SUBAPPLICATION FillWindowFS_AR (* Färbt ein FillAttributes-Objekt grün innerhalb [rWindowMin, rWindowMax], rot außerhalb (AR-Eingang) *)
  (* Standard: 61499-2; Description: Copyright (c) 2026 Meisterschulen am Ostbahnhof This program and the accompanying materials are made available under the terms of the Eclipse Public License 2.0 which is available at https://www.eclipse.org/legal/epl-2.0/ SPDX-License-Identifier: EPL-2.0 *)
  (* Version 2.0, 2026-09-11, Franz Höpfinger, Meisterschulen am Ostbahnhof, Umgebaut auf adapter::Engineering::measurements::AR_DEADBAND_COMPARE (jetzt allgemein fuer beliebige Fenster [WINDOW_MIN,WINDOW_MAX], nicht nur symmetrisches Totband) statt eigener Split/GE/LE/AND-Verdrahtung - CENTERED direkt als Gruen/Rot-Auswahl verwendet. *)
  (* Version 1.0, 2026-09-06, Franz Höpfinger, Meisterschulen am Ostbahnhof, initial API and implementation and/or initial documentation - built as a SubAppType (like MyLib_AX's GreenRedBackground1_AX) rather than a custom FBType with an ST helper function; a proper Q_FillAttributes adapter-wrapper FBType is a possible later refinement *)
  PACKAGE MyLib::sys;
  IMPORT isobus::UT::Q::Q_FillAttributes;
  IMPORT isobus::UT::Q::const::IDs::ID_NULL;
  IMPORT isobus::UT::Q::const::colours::COLOR_GREEN;
  IMPORT isobus::UT::Q::const::colours::COLOR_RED;
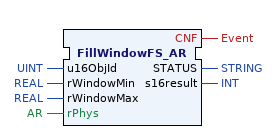
  EVENT_OUTPUT
    CNF; (* Confirmation of Requested Service *)
  END_EVENT
  VAR_INPUT
    u16ObjId : UINT := ID_NULL; (* FillAttributes object ID to command *)
    rWindowMin : REAL; (* Lower bound of the window that shows green *)
    rWindowMax : REAL; (* Upper bound of the window that shows green *)
  END_VAR
  VAR_OUTPUT
    STATUS : STRING; (* Service Status - passthrough from the internal Q_FillAttributes *)
    s16result : INT; (* retval - passthrough from the internal Q_FillAttributes *)
  END_VAR
  SOCKETS
    rPhys : adapter::types::unidirectional::AR; (* Value whose position relative to the window decides the colour *)
  END_SOCKETS
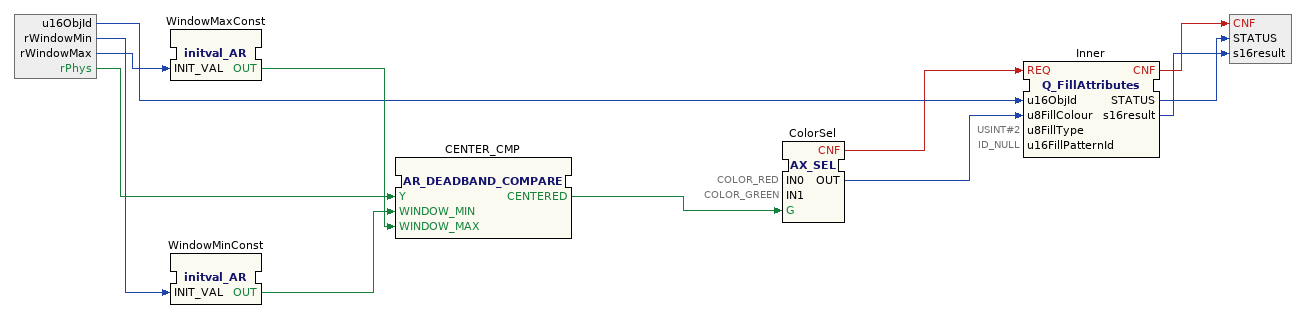
  FBS
    WindowMinConst : adapter::types::unidirectional::AR::initval::initval_AR;
    WindowMaxConst : adapter::types::unidirectional::AR::initval::initval_AR;
    CENTER_CMP : adapter::Engineering::measurements::AR_DEADBAND_COMPARE;
    ColorSel : adapter::iec61131::selection::AX_SEL(IN0 := COLOR_RED, IN1 := COLOR_GREEN);
    Inner : isobus::UT::Q::Q_FillAttributes(u8FillType := USINT#2, u16FillPatternId := ID_NULL);
  END_FBS
  EVENT_CONNECTIONS
    ColorSel.CNF TO Inner.REQ;
    Inner.CNF TO CNF;
  END_CONNECTIONS
  DATA_CONNECTIONS
    rWindowMin TO WindowMinConst.INIT_VAL;
    rWindowMax TO WindowMaxConst.INIT_VAL;
    u16ObjId TO Inner.u16ObjId;
    ColorSel.OUT TO Inner.u8FillColour;
    Inner.STATUS TO STATUS;
    Inner.s16result TO s16result;
  END_CONNECTIONS
  ADAPTER_CONNECTIONS
    rPhys TO CENTER_CMP.Y;
    WindowMinConst.OUT TO CENTER_CMP.WINDOW_MIN;
    WindowMaxConst.OUT TO CENTER_CMP.WINDOW_MAX;
    CENTER_CMP.CENTERED TO ColorSel.G;
  END_CONNECTIONS
END_SUBAPPLICATION
